(* IEC 61131-3 sources: generating_plc_code_with_llms/Code#2/ChatGPT_4/third run, 21 files *)

(* ---- 14.st ---- *)
// 60.89s
// 4
FUNCTION FC1001 : BOOL
VAR_INPUT
    MEW: REAL; // Measured value
    SP: REAL;  // Setpoint
    HYS: REAL; // Hysteresis in percentage of the setpoint
END_VAR
VAR_IN_OUT
    OUT: BOOL; // Output control
END_VAR
VAR
    P_HYS: REAL; // Hysteresis value
END_VAR

P_HYS := SP * HYS / 100.0; // Calculate hysteresis value

IF OUT THEN
    // Check if the measured value falls below the setpoint minus hysteresis
    IF MEW < (SP - P_HYS) THEN
        OUT := FALSE;
    END_IF;
ELSE
    // Check if the measured value exceeds the setpoint plus hysteresis
    IF MEW > (SP + P_HYS) THEN
        OUT := TRUE;
    END_IF;
END_IF;

FC1001 := OUT; // Set function return value
END_FUNCTION

(* ---- 15.st ---- *)
// 53.29s
// 4
FUNCTION FC1002 : BOOL
VAR_INPUT
    E_A : BOOL;      // Switch to turn on/off the monitoring system
    SENSOR : BOOL;   // Ultrasonic sensor input
    ZEITW : TIME;    // Time duration to switch from warning to alarm (e.g., T#3s for 3 seconds)
END_VAR
VAR_IN_OUT
    ZEIT : TON;      // Timer for tracking the duration of sensor perception
    P_HU, P_AL : BOOL; // Horn for warning and alarm outputs
END_VAR

IF E_A THEN
    // Monitoring system is turned on
    IF SENSOR THEN
        // Sensor detects something
        ZEIT(IN := TRUE, PT := ZEITW); // Start or continue the timer
        IF ZEIT.Q THEN
            // If perception lasts longer than ZEITW
            P_HU := FALSE; // Turn off horn
            P_AL := TRUE;  // Turn on alarm
        ELSE
            P_HU := TRUE;  // Turn on horn
        END_IF;
    ELSE
        // No detection by sensor
        ZEIT(IN := FALSE); // Stop the timer
        P_HU := FALSE;     // Turn off horn
    END_IF;
ELSE
    // Monitoring system is turned off
    ZEIT(IN := FALSE); // Stop the timer
    P_HU := FALSE;     // Turn off horn
    P_AL := FALSE;     // Turn off alarm
END_IF;

FC1002 := E_A; // Return the status of the monitoring system
END_FUNCTION

(* ---- 18.st ---- *)
// 30.75s
// 4
FUNCTION FC1003 : VOID
VAR_INPUT
    IN_R : REAL; // Input value
    IN_MAX, IN_MIN : REAL; // Input range
    OUT_MAX, OUT_MIN : REAL; // Output range
END_VAR
VAR_OUTPUT
    OUT_R : REAL; // Output value
    FEH : BOOL; // Error flag
END_VAR
VAR_TEMP
    DIFF1, DIFF2 : REAL;
END_VAR

// Check for valid input range to prevent division by zero
IF IN_MAX = IN_MIN THEN
    FEH := TRUE; // Set error flag if input range is invalid
    RETURN;
END_IF;

// Calculate the difference in the ranges
DIFF1 := IN_MAX - IN_MIN;
DIFF2 := OUT_MAX - OUT_MIN;

// Perform the linear scaling
OUT_R := OUT_MIN + (IN_R - IN_MIN) * DIFF2 / DIFF1;

FEH := FALSE; // Clear error flag if operation is successful
END_FUNCTION

(* ---- 19.st ---- *)
// 33.59s
// 4
FUNCTION_BLOCK FB1005
VAR_INPUT
    START : BOOL;       // Start/end signal for the measurement
    DICKE, V_MAX, V_MIN : REAL; // Thickness measurement and tolerance values
END_VAR
VAR_OUTPUT
    D_MAX, D_MIN : REAL; // Outputs for max and min thickness values
    P1 : BOOL;           // Output for reject light
END_VAR
VAR
    FO : BOOL;           // Flag for ongoing measurement
END_VAR

IF START THEN
    IF NOT FO THEN
        // New measurement cycle begins
        FO := TRUE; // Flag to indicate measurement is ongoing
        D_MAX := DICKE; // Initialize max and min values
        D_MIN := DICKE;
    ELSE
        // Update max and min values during the measurement
        IF DICKE > D_MAX THEN
            D_MAX := DICKE;
        END_IF;
        IF DICKE < D_MIN THEN
            D_MIN := DICKE;
        END_IF;
    END_IF;
ELSE
    IF FO THEN
        // Measurement cycle ends
        FO := FALSE; // Reset flag
        // Check if measured values are outside the tolerance range
        P1 := (D_MAX > V_MAX) OR (D_MIN < V_MIN);
    END_IF;
END_IF;
END_FUNCTION_BLOCK

(* ---- 20.st ---- *)
// 29.54s
// 3
FUNCTION_BLOCK INTERLOCK
VAR_INPUT
    I1 : BOOL;  // Input for controlling Q1
    I2 : BOOL;  // Input for controlling Q2
    TL : TIME;  // Dead time between outputs
END_VAR
VAR_OUTPUT
    Q1 : BOOL;  // Output 1
    Q2 : BOOL;  // Output 2
END_VAR
VAR
    T1 : TOF;   // Timer for Q1
    T2 : TOF;   // Timer for Q2
END_VAR

// Timer for Q1
T1(IN := NOT Q1, PT := TL);

// Timer for Q2
T2(IN := NOT Q2, PT := TL);

// Logic for Q1 and Q2 with interlock functionality
IF I1 AND NOT Q2 AND T2.Q THEN
    Q1 := TRUE;
ELSE
    Q1 := FALSE;
END_IF;

IF I2 AND NOT Q1 AND T1.Q THEN
    Q2 := TRUE;
ELSE
    Q2 := FALSE;
END_IF;

END_FUNCTION_BLOCK

(* ---- 21.st ---- *)
// 122.22s
// 4
FUNCTION_BLOCK BURNER
VAR_INPUT
    IN : BOOL;
    STAGE2 : BOOL;
    OVER_TEMP : BOOL;
    OIL_TEMP : BOOL := TRUE;
    FLAME : BOOL;
    RST : BOOL;
    RST_TIMER : BOOL;
    PRE_HEAT_TIME : TIME := T#5S;
    PRE_VENT_TIME : TIME := T#15S;
    PRE_IGNITE_TIME : TIME := T#15S;
    POST_IGNITE_TIME : TIME := T#25S;
    STAGE2_DELAY : TIME := T#10S;
    SAFETY_TIME : TIME := T#5S;
    LOCKOUT_TIME : TIME := T#10S;
    MULTIPLE_IGNITION : BOOL := TRUE;
    KW1 : REAL;
    KW2 : REAL;
END_VAR
VAR_OUTPUT
    MOTOR : BOOL;
    COIL1 : BOOL;
    COIL2 : BOOL;
    PRE_HEAT : BOOL;
    IGNITE : BOOL;
    FAIL : BOOL;
    KWH : REAL;
    STATUS : BYTE;
END_VAR
VAR_IN_OUT
    RUNTIME1 : UDINT;
    RUNTIME2 : UDINT;
    CYCLES : UDINT;
END_VAR
VAR
    state : INT;
    last_change : TIME;
    timer1 : TON;
    timer2 : TON;
    oil_temp_last : BOOL;
END_VAR

// Reset functionality
IF RST THEN
    state := 0; // Reset state to initial
    FAIL := FALSE;
    STATUS := 0;
    MOTOR := FALSE;
    COIL1 := FALSE;
    COIL2 := FALSE;
    PRE_HEAT := FALSE;
    IGNITE := FALSE;
END_IF;

// Over temperature check
IF OVER_TEMP THEN
    FAIL := TRUE;
    STATUS := 9; // Error code for over temperature
    RETURN;
END_IF;

// Main state machine for burner control
CASE state OF
    0:
        IF IN THEN
            PRE_HEAT := TRUE;
            timer1(IN := TRUE, PT := PRE_HEAT_TIME); // Start pre-heating timer
            state := 1;
            STATUS := 111; // Startup sequence
        ELSE
            STATUS := 110; // Wait for start signal (Standby)
        END_IF;
    1:
        IF NOT OIL_TEMP THEN
            IF timer1.Q THEN
                // Pre-heat time expired without reaching oil temp
                FAIL := TRUE;
                STATUS := 1; // Error code for fuel oil warming not responding
                state := 99; // Move to error state
            END_IF;
        ELSE
            MOTOR := TRUE; // Start motor and fan
            timer2(IN := TRUE, PT := PRE_VENT_TIME + PRE_IGNITE_TIME); // Start ignition timer
            state := 2; // Move to ignition state
        END_IF;
    2:
        IF timer2.ET >= PRE_VENT_TIME THEN
            IGNITE := TRUE;
            COIL1 := TRUE; // Open oil valve
            // Wait for flame or safety timer
            IF FLAME THEN
                state := 3; // Move to running state
                STATUS := 112; // Burner runs on stage 1
            ELSIF timer2.Q THEN
                // Safety time expired without flame
                FAIL := TRUE;
                STATUS := 4; // Error code for safety time expired without flame
                state := 99; // Move to error state
            END_IF;
        END_IF;
    // Additional states for stage 2, multiple ignition, and error handling could be added here
    99:
        // Error state
        MOTOR := FALSE;
        COIL1 := FALSE;
        COIL2 := FALSE;
        PRE_HEAT := FALSE;
        IGNITE := FALSE;
        // Lockout handling, resetting, and error messaging would be managed here
END_CASE;

// Update timers
timer1(IN := (state = 1) AND NOT OIL_TEMP, PT := PRE_HEAT_TIME);
timer2(IN := (state = 2), PT := PRE_VENT_TIME + PRE_IGNITE_TIME + SAFETY_TIME);
END_FUNCTION_BLOCK

(* ---- 1.st ---- *)
// 22.05s
// 4
VAR
	xAllOn : BOOL;
	xAllOff : BOOL;
	xAlarm1 : BOOL;
    xAlarm2 : BOOL;
END_VAR

// Main control logic
IF xAllOn THEN
    xAlarm1 := TRUE;
    xAlarm2 := TRUE;
    xAllOn := FALSE; // Turn off the signal after setting alarms
ELSIF xAllOff THEN
    xAlarm1 := FALSE;
    xAlarm2 := FALSE;
    xAllOff := FALSE; // Turn off the signal after resetting alarms
END_IF;

(* ---- 10.st ---- *)
// 24.24s
// 4
VAR_INPUT
    X : REAL; // Input to the sigmoid function
END_VAR

VAR
    Sigmoid : REAL; // Result of the sigmoid function
END_VAR

// Implementing the sigmoid function
Sigmoid := 1 / (1 + EXP(-X));

(* ---- 11.st ---- *)
// 23.42s
// 4
VAR_INPUT
    x : REAL; // Input value
END_VAR

VAR
    signResult : INT; // Result of the sign function
END_VAR

// Implementing the sign function
IF x < 0 THEN
    signResult := -1;
ELSIF x = 0 THEN
    signResult := 0;
ELSE
    signResult := 1;
END_IF;

(* ---- 12.st ---- *)
// 14.9s
// 4
VAR
    X : REAL; // Input value
    sinhX : REAL; // Result of hyperbolic sine function
END_VAR

// Implementing the hyperbolic sine function
sinhX := (EXP(X) - EXP(-X)) / 2;

(* ---- 13.st ---- *)
// 20.39s
// 2
VAR CONSTANT
    MAXNUMBERS : UINT := 99; // Index goes from 0 to 99 for 100 numbers
END_VAR

VAR
    aNumbers : ARRAY[0..MAXNUMBERS] OF INT; // Array of 100 random numbers
    nCnt : INT := 0; // Counter for the loop
END_VAR

// Initialize nCnt
nCnt := 0;

// Repeat loop to search through the array
REPEAT
    // Check if current number is 10
    IF aNumbers[nCnt] = 10 THEN
        EXIT; // Exit the loop if number is found
    END_IF;

    // Increment the counter
    nCnt := nCnt + 1;
UNTIL nCnt > MAXNUMBERS; // Continue until the end of the array is reached

(* ---- 16.st ---- *)
// 53.11s
// 4
VAR
    North_green : BOOL;
    North_yellow : BOOL;
    North_red : BOOL;
    East_green : BOOL;
    East_yellow : BOOL;
    East_red : BOOL;
    T1 : TON;
END_VAR

// Initialize and start the timer
T1(IN := TRUE, PT := T#10000ms);

// Logic for North light
North_green := T1.ET < T#5000ms;
North_yellow := T1.ET >= T#5000ms AND T1.ET < T#5500ms;
North_red := T1.ET >= T#5500ms;

// Logic for East light
East_green := T1.ET >= T#5500ms AND T1.ET < T#9500ms;
East_yellow := T1.ET >= T#9500ms AND T1.ET < T#10000ms;
East_red := T1.ET < T#5500ms OR T1.ET >= T#10000ms;

// Reset timer if it completes the cycle
IF T1.Q THEN
    T1.IN := FALSE; // Reset timer
    T1(IN := TRUE, PT := T#10000ms); // Restart timer
END_IF;

(* ---- 17.st ---- *)
// 28.12s
// 4
VAR
    aiOutside : INT; // Analog input for temperature (assumed scaled to °C)
    aiHumidity : INT; // Analog input for humidity (assumed scaled to %)
    sShowText : STRING[80]; // String to display the status
END_VAR

// Evaluating temperature and humidity
IF aiOutside < 18 THEN
    sShowText := 'Cold';
ELSIF aiOutside >= 18 AND aiOutside <= 25 THEN
    // Nested IF for humidity check within optimal temperature range
    IF aiHumidity >= 40 AND aiHumidity <= 75 THEN
        sShowText := 'Opt';
    ELSE
        sShowText := 'Temp. OK';
    END_IF;
ELSIF aiOutside > 25 THEN
    sShowText := 'Hot';
ELSE
    sShowText := 'Temp. OK'; // Default message in case of unexpected values
END_IF;

(* ---- 2.st ---- *)
// 24.85s
// 3
VAR_INPUT
    N : INT;
    K : INT;
END_VAR

VAR
    i : INT;
    N_Factorial : INT := 1; // N!
    K_Factorial : INT := 1; // K!
    NK_Factorial : INT := 1; // (N-K)!
    BinCoeff : INT; // Binomial Coefficient
END_VAR

// Calculate N!
FOR i := 1 TO N DO
    N_Factorial := N_Factorial * i;
END_FOR

// Calculate K!
FOR i := 1 TO K DO
    K_Factorial := K_Factorial * i;
END_FOR

// Calculate (N-K)!
FOR i := 1 TO N - K DO
    NK_Factorial := NK_Factorial * i;
END_FOR

// Calculate Binomial Coefficient: N! / (K! * (N-K)!)
BinCoeff := N_Factorial / (K_Factorial * NK_Factorial);

(* ---- 3.st ---- *)
// 21.82s
// 3
VAR_INPUT
    X : INT; // The position in the Fibonacci sequence
END_VAR

VAR
    t1 : DINT := 0; // First term
    t2 : DINT := 1; // Second term
    x_tmp : INT;
    i : INT;
    nextTerm : DINT;
END_VAR

IF X <= 0 THEN
    // Negative or zero index, not valid for Fibonacci sequence
    t1 := -1; // Indicate an error or invalid input
ELSIF X = 1 THEN
    t1 := 0; // First Fibonacci number is 0
ELSIF X = 2 THEN
    t1 := 1; // Second Fibonacci number is 1
ELSE
    FOR i := 3 TO X DO
        nextTerm := t1 + t2;
        t1 := t2;
        t2 := nextTerm;
    END_FOR
    t1 := nextTerm; // t1 now contains the Xth Fibonacci number
END_IF;

(* ---- 4.st ---- *)
// 26.36s
// 2
VAR
    aiLevel : INT;     // Analog input for fill level
    PercentLevel : UINT; // Converted fill level in percentage
    doLow : BOOL;      // Output for low fill level
    doOk : BOOL;       // Output for ok fill level
    doHigh : BOOL;     // Output for high fill level
    doAlarm : BOOL;    // Output for warning horn
END_VAR

// Convert analog input to percentage
PercentLevel := UINT((REAL(aiLevel) / 32767) * 100);

// Reset outputs
doLow := FALSE;
doOk := FALSE;
doHigh := FALSE;

// Check fill level and set outputs accordingly
CASE PercentLevel OF
    0..1:
    BEGIN
        doLow := TRUE;
        doAlarm := TRUE; // Activate alarm if level is below 1%
    END
    2..75:
    BEGIN
        doOk := TRUE;
    END
    76..100:
    BEGIN
        doHigh := TRUE;
    END
END_CASE;

(* ---- 5.st ---- *)
// 32.03s
// 3
VAR
    Start_Loop : BOOL := FALSE;
    one_hour : TIME := T#1h;
    One_Hour_Timer : TON;
    Gate_Open : BOOL := FALSE;
    Close_Gate_Inst : BOOL := FALSE;
    Sensed_Car : BOOL := FALSE;
    Sensed_Car_Inst : BOOL := FALSE;
    Sensed_App : BOOL := FALSE;
    Mobile_Inst : BOOL := FALSE;
    Auth : STRING;
    my_defined_str : STRING := 'abcd';
END_VAR

// Timer control
IF NOT Start_Loop THEN
    One_Hour_Timer(IN := TRUE, PT := one_hour);
ELSE
    One_Hour_Timer(IN := FALSE);
END_IF;

// Check if timer has timed out and the gate is open
IF One_Hour_Timer.Q AND Gate_Open THEN
    Close_Gate_Inst := TRUE; // Instruction to close the gate
    Gate_Open := FALSE; // Gate is now closed
ELSE
    Close_Gate_Inst := FALSE;
END_IF;

// Check for car or app and validate authentication
IF (Sensed_Car OR Sensed_App) AND (Auth = my_defined_str) THEN
    Gate_Open := TRUE; // Open the gate
ELSE
    Sensed_Car_Inst := FALSE;
    Mobile_Inst := FALSE;
END_IF;

(* ---- 6.st ---- *)
// 45.5s
// 2
VAR CONSTANT
    WAIT : UINT:= 0;
    TOP_POSITION : UINT:= 1;
    BOTTOM_POSITION : UINT:= 2;
    GETBOX : UINT:= 3;
    UNLOAD_POSITION : UINT:= 4;
    UNLOAD_BOX : UINT:= 5;
END_VAR

VAR
    doConvTop: BOOL;
    doConvBottom: BOOL;
    doConvLift: BOOL;
    doLiftTop: BOOL;
    doLiftBottom: BOOL;
    doLiftUnload: BOOL;
    diConvTop: BOOL;
    diConvBottom: BOOL;
    diLiftTop: BOOL;
    diLiftBottom: BOOL;
    diLiftUnload: BOOL;
    diBoxLift: BOOL;
    selectLift: UINT := WAIT;
    ConvTopOn: BOOL;
    ConvBottomOn: BOOL;
END_VAR

// Control Logic
CASE selectLift OF
    WAIT:
    BEGIN
        IF diConvTop THEN
            doConvTop := FALSE;
            selectLift := TOP_POSITION;
        ELSIF diConvBottom THEN
            doConvBottom := FALSE;
            selectLift := BOTTOM_POSITION;
        END_IF;
    END

    TOP_POSITION:
    BEGIN
        doLiftTop := TRUE;
        doLiftBottom := FALSE;
        IF diLiftTop THEN
            doConvLift := TRUE;
            selectLift := GETBOX;
        END_IF;
    END

    BOTTOM_POSITION:
    BEGIN
        doLiftBottom := TRUE;
        doLiftTop := FALSE;
        IF diLiftBottom THEN
            doConvLift := TRUE;
            selectLift := GETBOX;
        END_IF;
    END

    GETBOX:
    BEGIN
        IF diBoxLift THEN
            doConvLift := FALSE;
            selectLift := UNLOAD_POSITION;
        END_IF;
    END

    UNLOAD_POSITION:
    BEGIN
        doLiftUnload := TRUE;
        IF diLiftUnload THEN
            selectLift := UNLOAD_BOX;
        END_IF;
    END

    UNLOAD_BOX:
    BEGIN
        // Assuming there's an output to control unloading conveyor (not specified in VAR)
        // doUnloadingConveyor := TRUE;
        // Reset lift position and unload flag after the box has left
        IF NOT diBoxLift THEN
            doLiftUnload := FALSE;
            selectLift := WAIT;
        END_IF;
    END
END_CASE;

(* ---- 7.st ---- *)
// 17.66s
// 2
VAR CONSTANT
    MAX_INDEX: USINT := 4; // 5 load receptors, indexed 0 to 4
END_VAR

VAR
    aWeights : ARRAY[0..MAX_INDEX] OF INT; // Array of weights from load receptors
    iCnt : USINT; // Counter for the loop
    sumWeight : DINT := 0; // Sum of weights
    avgWeight : INT; // Average weight
END_VAR

// Reset sumWeight
sumWeight := 0;

// Calculate the total weight
FOR iCnt := 0 TO MAX_INDEX DO
    sumWeight := sumWeight + aWeights[iCnt];
END_FOR;

// Calculate the average weight
avgWeight := INT(sumWeight / (MAX_INDEX + 1)); // Adding 1 since index starts from 0

(* ---- 8.st ---- *)
// 29.42s
// 2
VAR_INPUT
    X : REAL; // Input for the Lambert W function
END_VAR

VAR
    w : REAL := 0; // Initial guess for W(x)
    i : INT; // Counter for the loop
    we : REAL; // w * exp(w)
    w1e : REAL; // (w + 1) * exp(w)
    ewx : REAL; // exp(w) - x/w
    last : DWORD; // Last value of w for convergence check
END_VAR

// Iterative approximation using Newton's method
FOR i := 1 TO 100 DO // Limiting iterations to 100 for convergence
    we := w * EXP(w);
    w1e := (w + 1) * EXP(w);
    ewx := (we - X) / w1e;

    // Update w
    w := w - ewx;

    // Check for convergence
    IF DWORD(TO_REAL(w)) = last THEN
        EXIT; // Convergence achieved
    END_IF;
    last := DWORD(TO_REAL(w));
END_FOR;

(* ---- 9.st ---- *)
// 20.46s
// 4
VAR
    YEAR : INT; // Input Year
    IsLeapYear : BOOL; // Output: TRUE if leap year, FALSE otherwise
END_VAR

// Check if the year is a leap year
IsLeapYear := FALSE; // Default to false

IF (YEAR MOD 4 = 0) THEN
    IF (YEAR MOD 100 = 0) THEN
        IF (YEAR MOD 400 = 0) THEN
            IsLeapYear := TRUE; // Leap year if divisible by 400
        END_IF;
    ELSE
        IsLeapYear := TRUE; // Leap year if divisible by 4 but not by 100
    END_IF;
END_IF;
